{attribute 'qualified_only'}
{attribute 'strict'}
TYPE Rotation :
(
	UP := 0,
	RIGHT := 1,
	DOWN := 2,
	LEFT := 3
)DINT;
END_TYPE

(* stored: Version 1.1.0.1
   DUT Rotation: Id {26b50a4d-ba6d-4d89-b0e6-b79d7f82d566} *)
